FUNCTION_BLOCK FB_Frames
VAR_INPUT
END_VAR
VAR_OUTPUT
END_VAR
VAR
	AllFrames : ARRAY[0..40] OF Frame;
	ArrangedFrames : ARRAY[0..60] OF Frame;
	i: INT;
END_VAR

METHOD Map : ARRAY[0..60] OF Frame
VAR_INPUT
	aFrameString : ARRAY[0..60] OF STRING;
END_VAR
VAR
	i : INT;
	j : INT;
	PlaceHolder : ARRAY[0..60] OF Frame;
END_VAR
FOR i := 0 TO 60 DO
	IF aFrameString[i] = '' THEN
		PlaceHolder[i].Name := ''; 
		PlaceHolder[i].X := 0; 
		PlaceHolder[i].Y := 0; 
	ELSE
		FOR j := 0 TO 60 DO
			IF aFrameString[i] = AllFrames[j].Name THEN
				PlaceHolder[i] := AllFrames[j];
			ELSIF AllFrames[j].Name = '' THEN
				EXIT;
			END_IF
		END_FOR
		j := 0;
	END_IF
END_FOR
ArrangedFrames := PlaceHolder;
Map := PlaceHolder;
END_METHOD

METHOD Teach : BOOL
VAR_INPUT
	sName : STRING;
	rX : REAL;
	rY : REAL;
END_VAR
VAR
	i : INT;
END_VAR
FOR i := 0 TO 30 BY 1 DO
	IF AllFrames[i].Name = '' AND AllFrames[i].X = 0 AND AllFrames[i].Y = 0 THEN
		AllFrames[i].Name := sName;
		AllFrames[i].X := rX;
		AllFrames[i].Y := rY;
		Teach := TRUE;
		EXIT;
	END_IF
END_FOR
END_METHOD

END_FUNCTION_BLOCK

(* stored: Version 1.1.0.1, ProductVersion 3.1.4024.11
   POU FB_Frames: Id {ad93ff7e-d8a3-4bf2-8978-b19a0709c4ac}, SpecialFunc None
   Method Map: Id {459687c9-10ed-4392-89f1-e3d34977b4ca}
   Method Teach: Id {a56573b6-5505-4e7f-b46e-8b3a1e58c13e} *)
